TYPE ST_SelectorSwitchIO :
STRUCT
	Left	AT%I* :BIT;
	Right	AT%I* :BIT;	
END_STRUCT
END_TYPE

(* stored: Version 1.1.0.1, ProductVersion 3.1.4026.19
   DUT ST_SelectorSwitchIO: Id {54310838-d6d2-48c8-a7bb-6c18e15ba57b} *)
